(* PLC project SafeLOGIC-1, BrAutomation SafeDESIGNER  4.3.4.4 *)
(* stored: companyURL http://www.br-automation.com, creationDateTime Thu Sep 10 10:20:45 2020 *)

PROGRAM Main

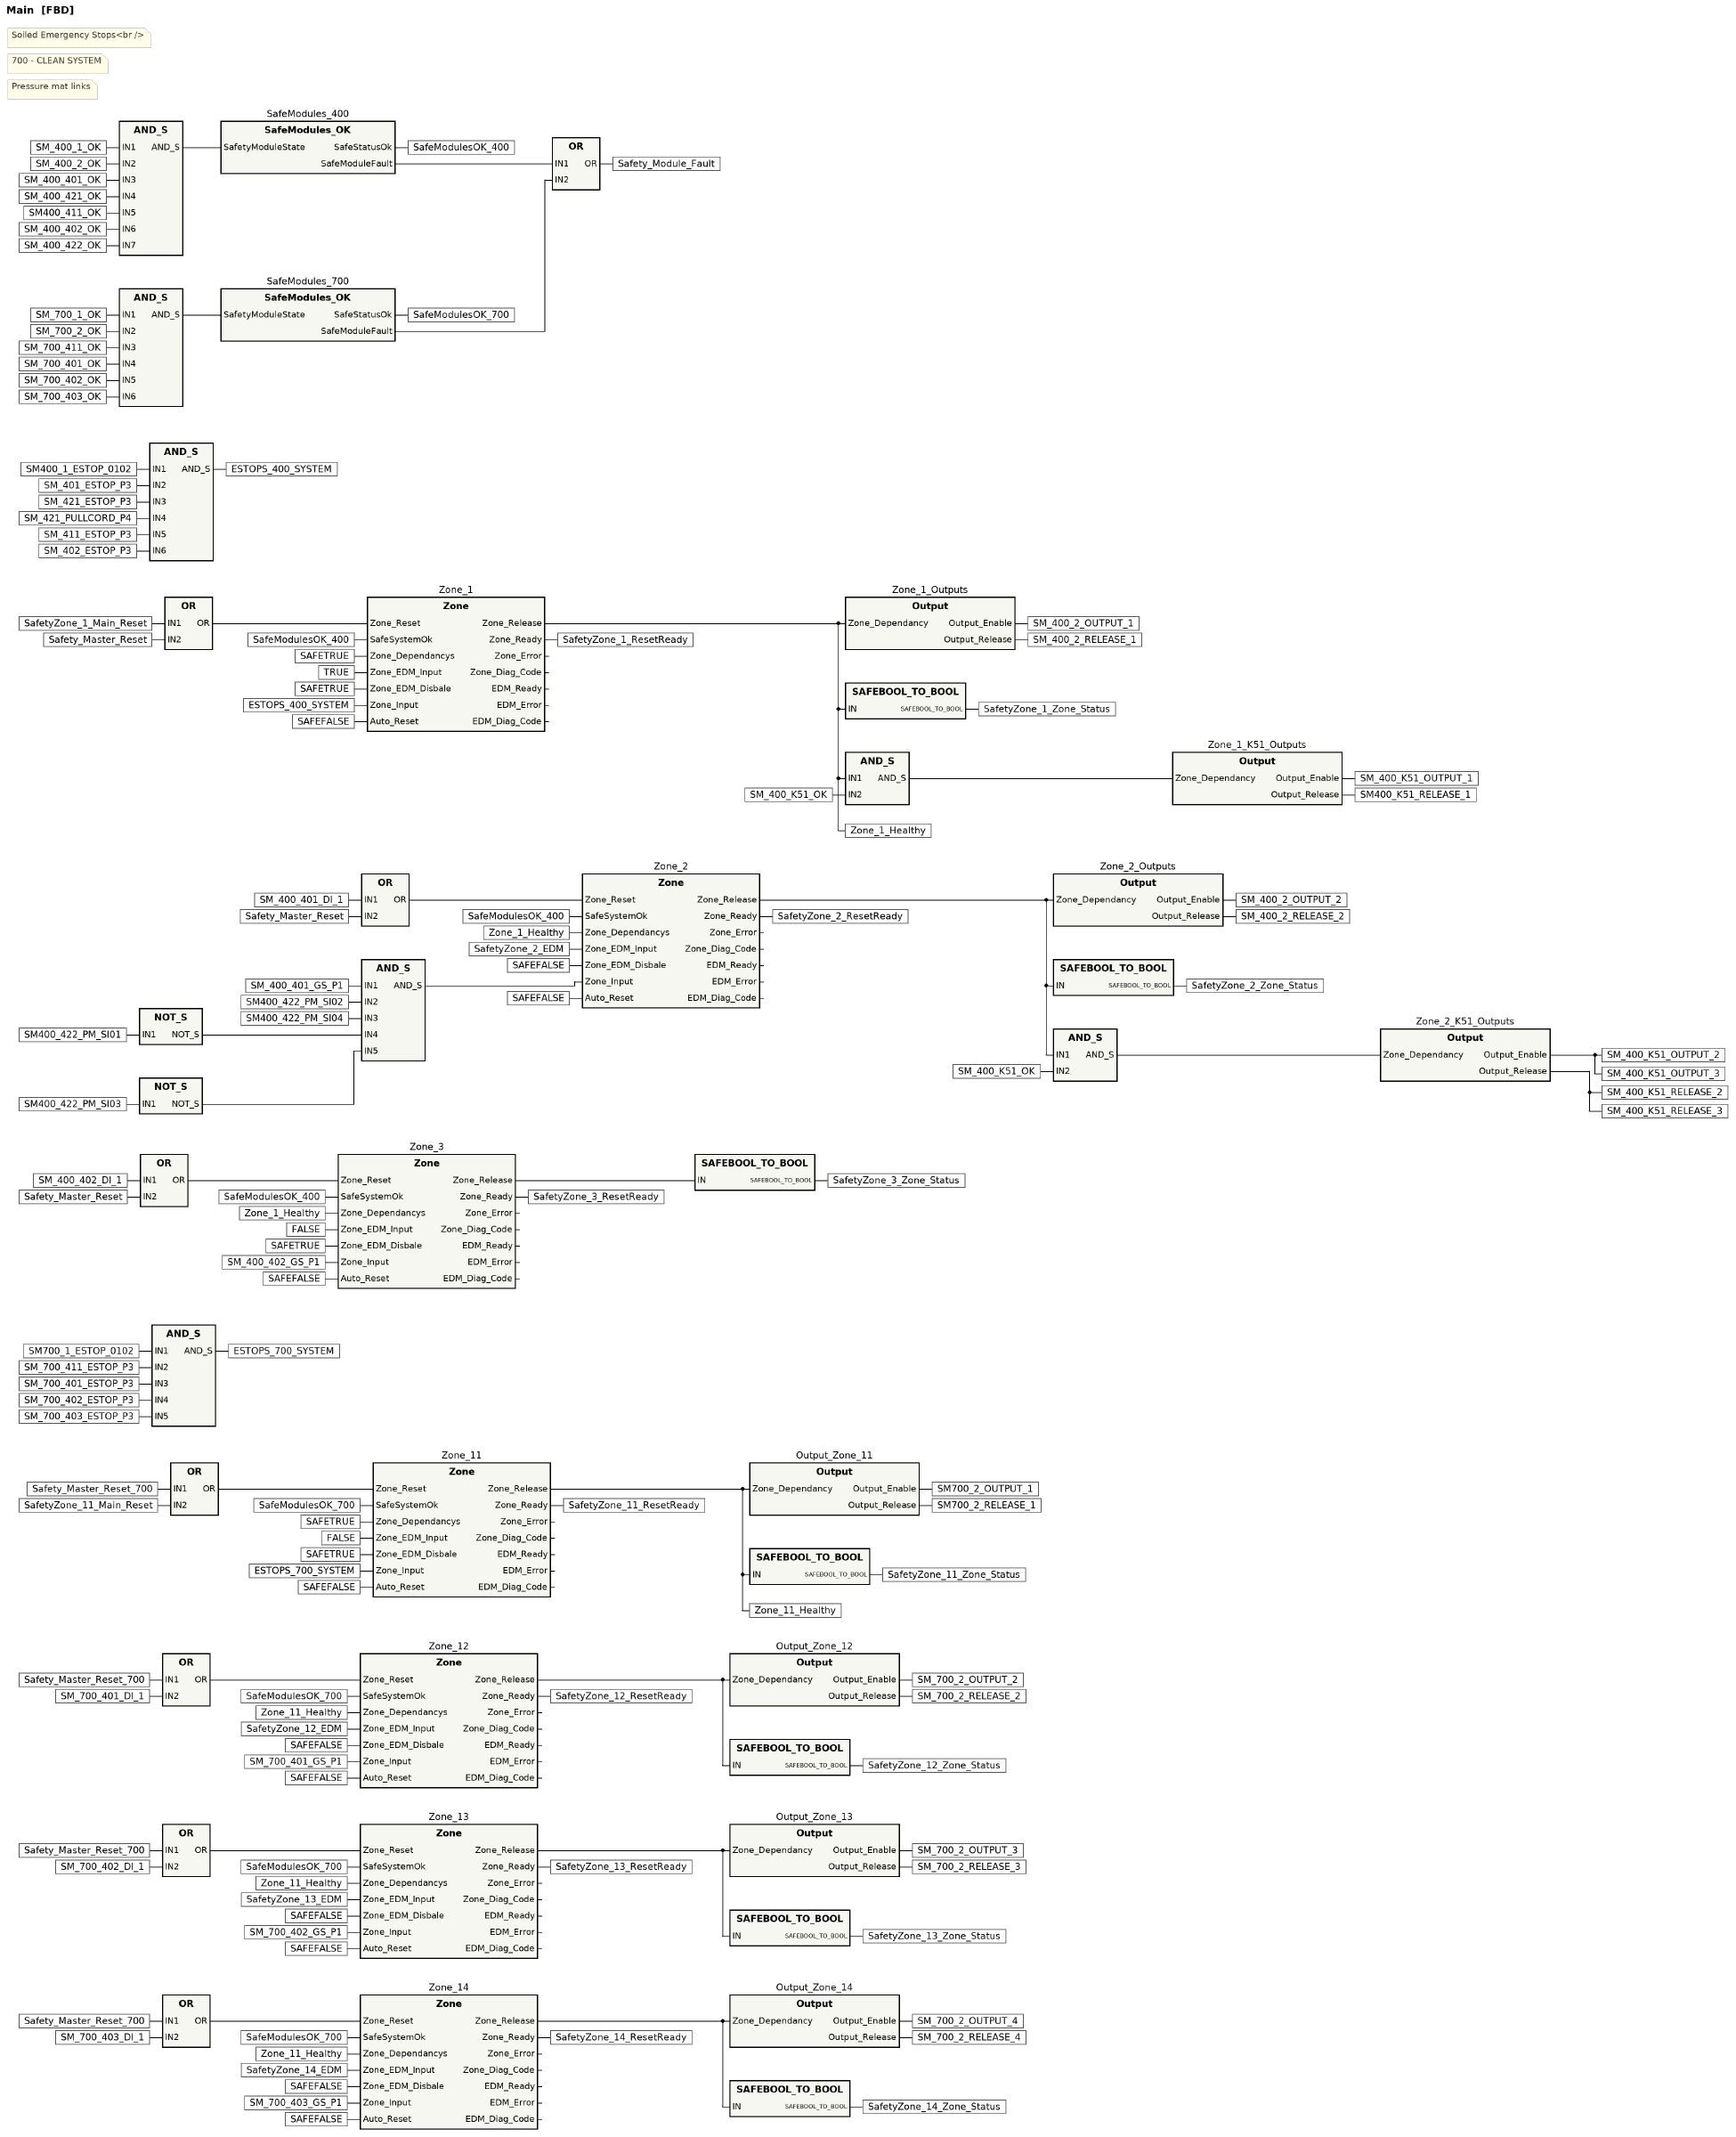
(* FBD diagram, written out as Structured Text *)
SafeModules_400(SafetyModuleState := AND_S(SM_400_1_OK, SM_400_2_OK, SM_400_401_OK, SM_400_421_OK, SM400_411_OK, SM_400_402_OK, SM_400_422_OK));
SafeModulesOK_400 := SafeModules_400.SafeStatusOk;
SafeModules_700(SafetyModuleState := AND_S(SM_700_1_OK, SM_700_2_OK, SM_700_411_OK, SM_700_401_OK, SM_700_402_OK, SM_700_403_OK));
SafeModulesOK_700 := SafeModules_700.SafeStatusOk;
Safety_Module_Fault := SafeModules_400.SafeModuleFault OR SafeModules_700.SafeModuleFault;
(* Soiled Emergency Stops<br /> *)
ESTOPS_400_SYSTEM := AND_S(SM400_1_ESTOP_0102, SM_401_ESTOP_P3, SM_421_ESTOP_P3, SM_421_PULLCORD_P4, SM_411_ESTOP_P3, SM_402_ESTOP_P3);
Zone_1(Zone_Reset := SafetyZone_1_Main_Reset OR Safety_Master_Reset, SafeSystemOk := SafeModulesOK_400, Zone_Dependancys := SAFETRUE, Zone_EDM_Input := TRUE, Zone_EDM_Disbale := SAFETRUE, Zone_Input := ESTOPS_400_SYSTEM, Auto_Reset := SAFEFALSE);
SafetyZone_1_Zone_Status := SAFEBOOL_TO_BOOL(Zone_1.Zone_Release);
Zone_1_Healthy := Zone_1.Zone_Release;
SafetyZone_1_ResetReady := Zone_1.Zone_Ready;
Zone_1_Outputs(Zone_Dependancy := Zone_1.Zone_Release);
SM_400_2_OUTPUT_1 := Zone_1_Outputs.Output_Enable;
SM_400_2_RELEASE_1 := Zone_1_Outputs.Output_Release;
Zone_1_K51_Outputs(Zone_Dependancy := AND_S(Zone_1.Zone_Release, SM_400_K51_OK));
SM_400_K51_OUTPUT_1 := Zone_1_K51_Outputs.Output_Enable;
SM400_K51_RELEASE_1 := Zone_1_K51_Outputs.Output_Release;
Zone_2(Zone_Reset := SM_400_401_DI_1 OR Safety_Master_Reset, SafeSystemOk := SafeModulesOK_400, Zone_Dependancys := Zone_1_Healthy, Zone_EDM_Input := SafetyZone_2_EDM, Zone_EDM_Disbale := SAFEFALSE, Zone_Input := AND_S(SM_400_401_GS_P1, SM400_422_PM_SI02, SM400_422_PM_SI04, NOT_S(SM400_422_PM_SI01), NOT_S(SM400_422_PM_SI03)), Auto_Reset := SAFEFALSE);
SafetyZone_2_ResetReady := Zone_2.Zone_Ready;
SafetyZone_2_Zone_Status := SAFEBOOL_TO_BOOL(Zone_2.Zone_Release);
Zone_2_Outputs(Zone_Dependancy := Zone_2.Zone_Release);
SM_400_2_OUTPUT_2 := Zone_2_Outputs.Output_Enable;
(* Pressure mat links *)
Zone_2_K51_Outputs(Zone_Dependancy := AND_S(Zone_2.Zone_Release, SM_400_K51_OK));
SM_400_K51_OUTPUT_3 := Zone_2_K51_Outputs.Output_Enable;
SM_400_2_RELEASE_2 := Zone_2_Outputs.Output_Release;
SM_400_K51_OUTPUT_2 := Zone_2_K51_Outputs.Output_Enable;
SM_400_K51_RELEASE_3 := Zone_2_K51_Outputs.Output_Release;
SM_400_K51_RELEASE_2 := Zone_2_K51_Outputs.Output_Release;
Zone_3(Zone_Reset := SM_400_402_DI_1 OR Safety_Master_Reset, SafeSystemOk := SafeModulesOK_400, Zone_Dependancys := Zone_1_Healthy, Zone_EDM_Input := FALSE, Zone_EDM_Disbale := SAFETRUE, Zone_Input := SM_400_402_GS_P1, Auto_Reset := SAFEFALSE);
SafetyZone_3_ResetReady := Zone_3.Zone_Ready;
SafetyZone_3_Zone_Status := SAFEBOOL_TO_BOOL(Zone_3.Zone_Release);
(* 700 - CLEAN SYSTEM *)
ESTOPS_700_SYSTEM := AND_S(SM700_1_ESTOP_0102, SM_700_411_ESTOP_P3, SM_700_401_ESTOP_P3, SM_700_402_ESTOP_P3, SM_700_403_ESTOP_P3);
Zone_11(Zone_Reset := Safety_Master_Reset_700 OR SafetyZone_11_Main_Reset, SafeSystemOk := SafeModulesOK_700, Zone_Dependancys := SAFETRUE, Zone_EDM_Input := FALSE, Zone_EDM_Disbale := SAFETRUE, Zone_Input := ESTOPS_700_SYSTEM, Auto_Reset := SAFEFALSE);
Zone_11_Healthy := Zone_11.Zone_Release;
SafetyZone_11_Zone_Status := SAFEBOOL_TO_BOOL(Zone_11.Zone_Release);
SafetyZone_11_ResetReady := Zone_11.Zone_Ready;
Output_Zone_11(Zone_Dependancy := Zone_11.Zone_Release);
SM700_2_OUTPUT_1 := Output_Zone_11.Output_Enable;
SM700_2_RELEASE_1 := Output_Zone_11.Output_Release;
Zone_12(Zone_Reset := Safety_Master_Reset_700 OR SM_700_401_DI_1, SafeSystemOk := SafeModulesOK_700, Zone_Dependancys := Zone_11_Healthy, Zone_EDM_Input := SafetyZone_12_EDM, Zone_EDM_Disbale := SAFEFALSE, Zone_Input := SM_700_401_GS_P1, Auto_Reset := SAFEFALSE);
SafetyZone_12_Zone_Status := SAFEBOOL_TO_BOOL(Zone_12.Zone_Release);
SafetyZone_12_ResetReady := Zone_12.Zone_Ready;
Output_Zone_12(Zone_Dependancy := Zone_12.Zone_Release);
SM_700_2_OUTPUT_2 := Output_Zone_12.Output_Enable;
SM_700_2_RELEASE_2 := Output_Zone_12.Output_Release;
Zone_13(Zone_Reset := Safety_Master_Reset_700 OR SM_700_402_DI_1, SafeSystemOk := SafeModulesOK_700, Zone_Dependancys := Zone_11_Healthy, Zone_EDM_Input := SafetyZone_13_EDM, Zone_EDM_Disbale := SAFEFALSE, Zone_Input := SM_700_402_GS_P1, Auto_Reset := SAFEFALSE);
SafetyZone_13_Zone_Status := SAFEBOOL_TO_BOOL(Zone_13.Zone_Release);
SafetyZone_13_ResetReady := Zone_13.Zone_Ready;
Output_Zone_13(Zone_Dependancy := Zone_13.Zone_Release);
SM_700_2_OUTPUT_3 := Output_Zone_13.Output_Enable;
SM_700_2_RELEASE_3 := Output_Zone_13.Output_Release;
Zone_14(Zone_Reset := Safety_Master_Reset_700 OR SM_700_403_DI_1, SafeSystemOk := SafeModulesOK_700, Zone_Dependancys := Zone_11_Healthy, Zone_EDM_Input := SafetyZone_14_EDM, Zone_EDM_Disbale := SAFEFALSE, Zone_Input := SM_700_403_GS_P1, Auto_Reset := SAFEFALSE);
SafetyZone_14_Zone_Status := SAFEBOOL_TO_BOOL(Zone_14.Zone_Release);
SafetyZone_14_ResetReady := Zone_14.Zone_Ready;
Output_Zone_14(Zone_Dependancy := Zone_14.Zone_Release);
SM_700_2_OUTPUT_4 := Output_Zone_14.Output_Enable;
SM_700_2_RELEASE_4 := Output_Zone_14.Output_Release;
END_PROGRAM
